ABB RobotStudio station: OefenenPad.rsstnx

Station OefenenPad (saved by RobotStudio 23.3.10550.0)
Controller IRB120_3_58
  mechanical unit ROB_1: IRB120_3_58__01, 6 joints, base frame (0, 0, 0) mm
Layout (positions relative to the parent item):
  - IRB120_3_58__01 [mechanism, from %ABB.RobotStudio.Models.IRB120%\IRB120_3_58_G_01.rslib] at (0, 0, 0) mm; joint values [0, -0.8728, 0.5337, 0, 0.8627, 0] (rad or m)
  - Table [part] at (200, -200, 0) mm, size 250 x 375 x 200 mm
  - MyTool_2 [mechanism, from Training Objects\myTool.rslib] at (117.02, 0, 594) mm, rotated rx 180 ry 60 rz 180 deg
Attachment: MyTool_2 is attached to IRB120_3_58__01 / Link6
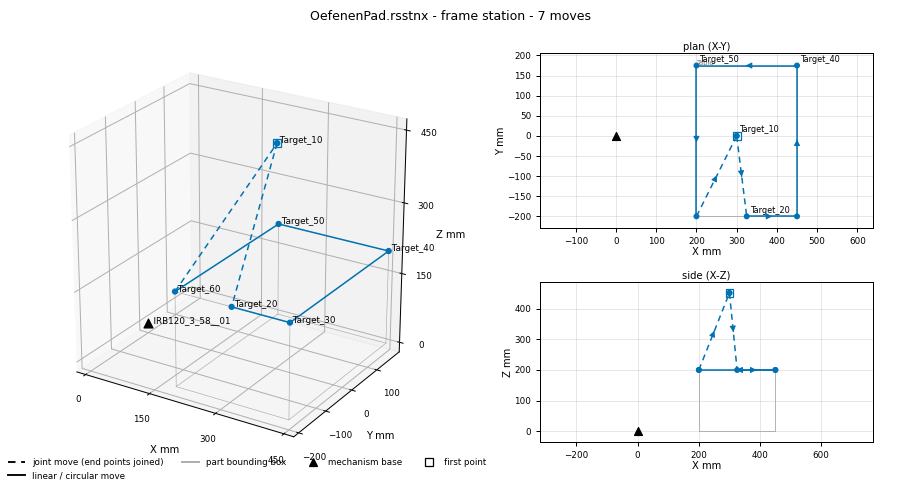
[picture p0: tool path of OefenenPad.rsstnx in frame station, 7 of 7 moves have a stored position in this frame; points joined in program order, loops and branches not executed]
Targets, tools, work objects and paths stored in the station, written as RAPID:
! task T_ROB1
MODULE CalibData
  PERS tooldata MyTool:=[TRUE,[[31.792631019,0,229.638935148],[0.945518576,0,0.325568154,0]],[1,[0,0,1],[1,0,0,0],0,0,0]];
  TASK PERS wobjdata wTable:=[FALSE,TRUE,"",[[0,0,0],[1,0,0,0]],[[200,-200,200],[1,0,0,0]]];
ENDMODULE

! task T_ROB1
MODULE MainModule
  CONST robtarget Target_10:=[[100.000062522,200,251.649955505],[0.19080893,0,0.981627196,0],[0,0,0,0],[9E+09,9E+09,9E+09,9E+09,9E+09,9E+09]];
  CONST robtarget Target_20:=[[125.000018184,-0.000019803,-0.00005763],[-0.000000057,0,1,-0.000000008],[-1,0,-1,0],[9E+09,9E+09,9E+09,9E+09,9E+09,9E+09]];
  CONST robtarget Target_30:=[[250.000014402,-0.000029072,-0.000060381],[-0.000000057,-0.000000012,1,-0.000000034],[-1,0,-1,0],[9E+09,9E+09,9E+09,9E+09,9E+09,9E+09]];
  CONST robtarget Target_40:=[[250.000017577,375.00000237,-0.000062564],[-0.000000056,-0.000000008,1,-0.000000008],[0,-1,0,0],[9E+09,9E+09,9E+09,9E+09,9E+09,9E+09]];
  CONST robtarget Target_50:=[[0.000024809,375.000009487,-0.000060256],[-0.00000005,-0.000000025,1,-0.000000022],[0,-1,1,0],[9E+09,9E+09,9E+09,9E+09,9E+09,9E+09]];
  CONST robtarget Target_60:=[[0.000025666,0.000095996,-0.001059984],[-0.000000743,-0.000000057,1,0.000000132],[-1,0,-2,0],[9E+09,9E+09,9E+09,9E+09,9E+09,9E+09]];
  CONST robtarget Target_70:=[[100.000153067,200,251.649947919],[0.190808843,0,0.981627213,0],[0,0,0,0],[9E+09,9E+09,9E+09,9E+09,9E+09,9E+09]];
  PROC Path_10()
    MoveJ Target_10,v1000,z100,MyTool\WObj:=wTable;
    MoveJ Target_20,v1000,z100,MyTool\WObj:=wTable;
    MoveL Target_30,v1000,z100,MyTool\WObj:=wTable;
    MoveL Target_40,v1000,z100,MyTool\WObj:=wTable;
    MoveL Target_50,v1000,z100,MyTool\WObj:=wTable;
    MoveL Target_60,v1000,z100,MyTool\WObj:=wTable;
    MoveJ Target_70,v1000,z100,MyTool\WObj:=wTable;
  ENDPROC
ENDMODULE

